FUNCTION FuzzyOR_array : real
VAR_INPUT
	ORmethod:eOrMethod;
END_VAR
VAR_IN_OUT
	Inputs:ARRAY[*]OF REAL;
END_VAR

VAR
	i: DINT;
END_VAR

FuzzyOR_array:=0;
FOR i:=LOWER_BOUND(Inputs,1) TO UPPER_BOUND(Inputs,1) DO
	IF inputs[i] > FuzzyOR_array THEN
		FuzzyOR_array := inputs[i];
	END_IF
END_FOR

END_FUNCTION

(* stored: Version 1.1.0.1, ProductVersion 3.1.4024.6
   POU FuzzyOR_array: Id {c5e3b8d3-a4a0-4344-abd8-e66584166d8f}, SpecialFunc None *)
